// Mitsubishi GX Works2 project: exam_practice   PLC: Q02/Q02H

PROGRAM Q5-MC
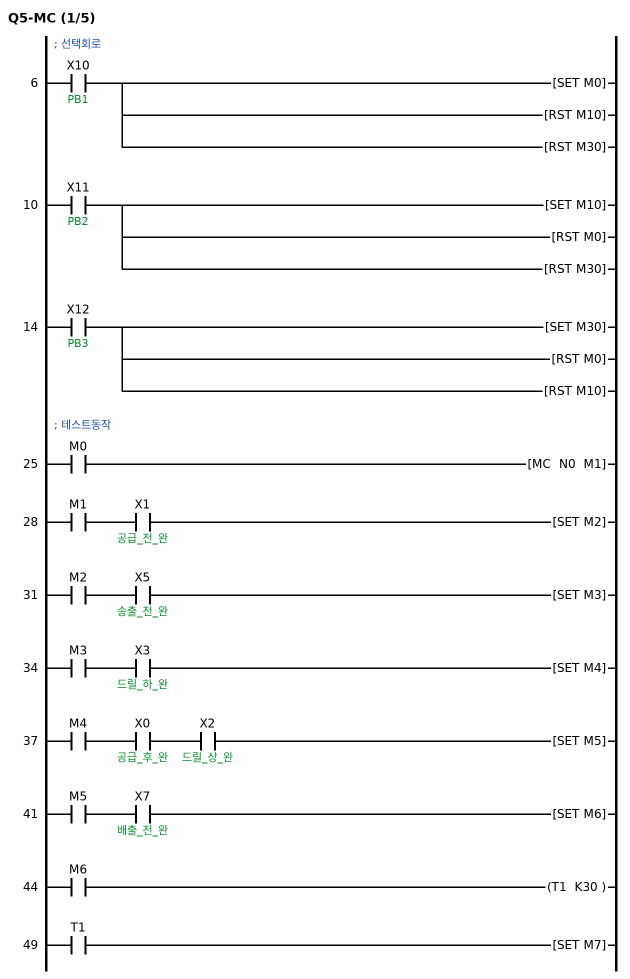
; 선택회로
6     LD      X10  ; PB1
      SET     M0
      RST     M10
      RST     M30
10    LD      X11  ; PB2
      SET     M10
      RST     M0
      RST     M30
14    LD      X12  ; PB3
      SET     M30
      RST     M0
      RST     M10
; 테스트동작
25    LD      M0
      MC      N0 M1
28    LD      M1
      AND     X1  ; 공급_전_완
      SET     M2
31    LD      M2
      AND     X5  ; 송출_전_완
      SET     M3
34    LD      M3
      AND     X3  ; 드릴_하_완
      SET     M4
37    LD      M4
      AND     X0  ; 공급_후_완
      AND     X2  ; 드릴_상_완
      SET     M5
41    LD      M5
      AND     X7  ; 배출_전_완
      SET     M6
44    LD      M6
      OUT     T1 K30
49    LD      T1
      SET     M7
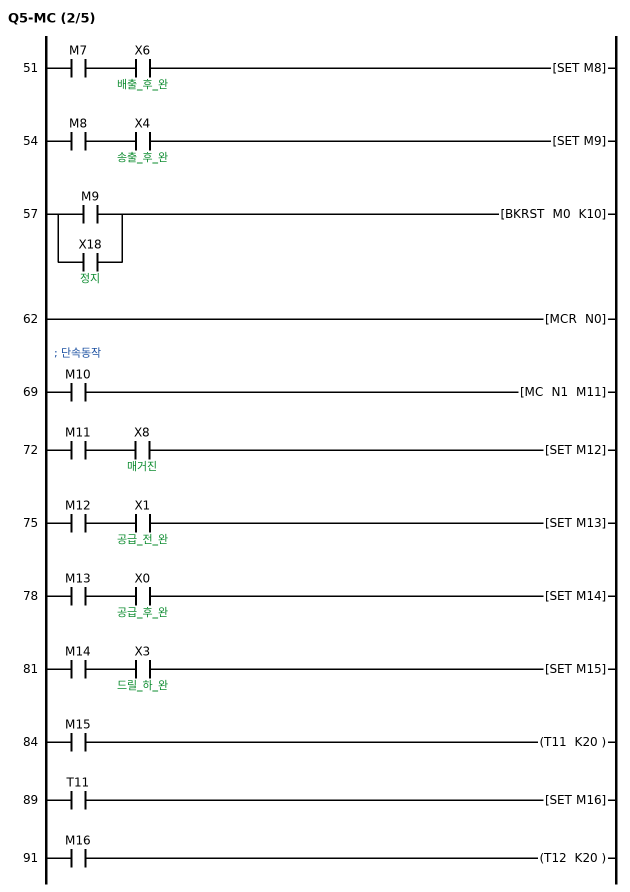
51    LD      M7
      AND     X6  ; 배출_후_완
      SET     M8
54    LD      M8
      AND     X4  ; 송출_후_완
      SET     M9
57    LD      M9
      OR      X18  ; 정지
      BKRST   M0 K10
62    MCR     N0
; 단속동작
69    LD      M10
      MC      N1 M11
72    LD      M11
      AND     X8  ; 매거진
      SET     M12
75    LD      M12
      AND     X1  ; 공급_전_완
      SET     M13
78    LD      M13
      AND     X0  ; 공급_후_완
      SET     M14
81    LD      M14
      AND     X3  ; 드릴_하_완
      SET     M15
84    LD      M15
      OUT     T11 K20
89    LD      T11
      SET     M16
91    LD      M16
      OUT     T12 K20
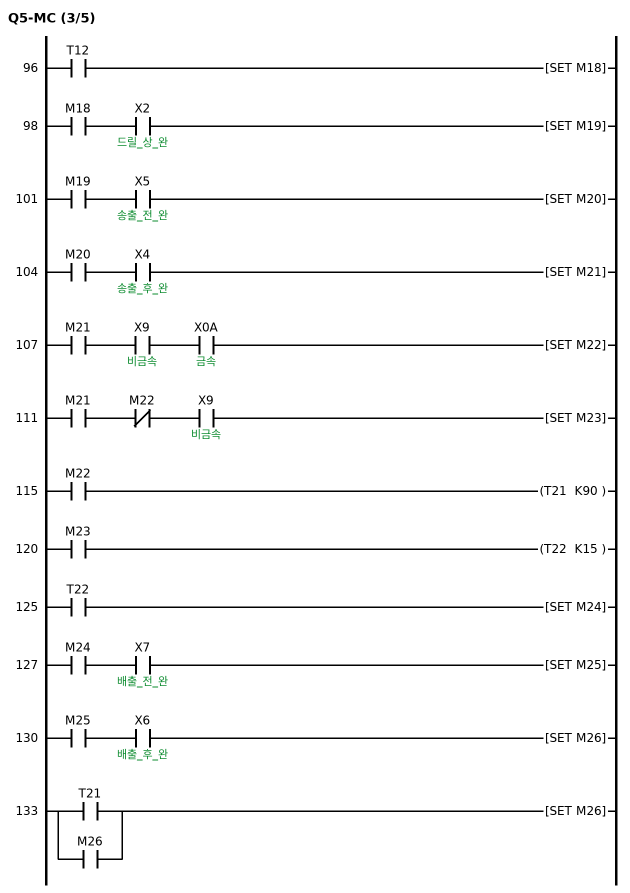
96    LD      T12
      SET     M18
98    LD      M18
      AND     X2  ; 드릴_상_완
      SET     M19
101   LD      M19
      AND     X5  ; 송출_전_완
      SET     M20
104   LD      M20
      AND     X4  ; 송출_후_완
      SET     M21
107   LD      M21
      AND     X9  ; 비금속
      AND     X0A  ; 금속
      SET     M22
111   LD      M21
      ANI     M22
      AND     X9  ; 비금속
      SET     M23
115   LD      M22
      OUT     T21 K90
120   LD      M23
      OUT     T22 K15
125   LD      T22
      SET     M24
127   LD      M24
      AND     X7  ; 배출_전_완
      SET     M25
130   LD      M25
      AND     X6  ; 배출_후_완
      SET     M26
133   LD      T21
      OR      M26
      SET     M26
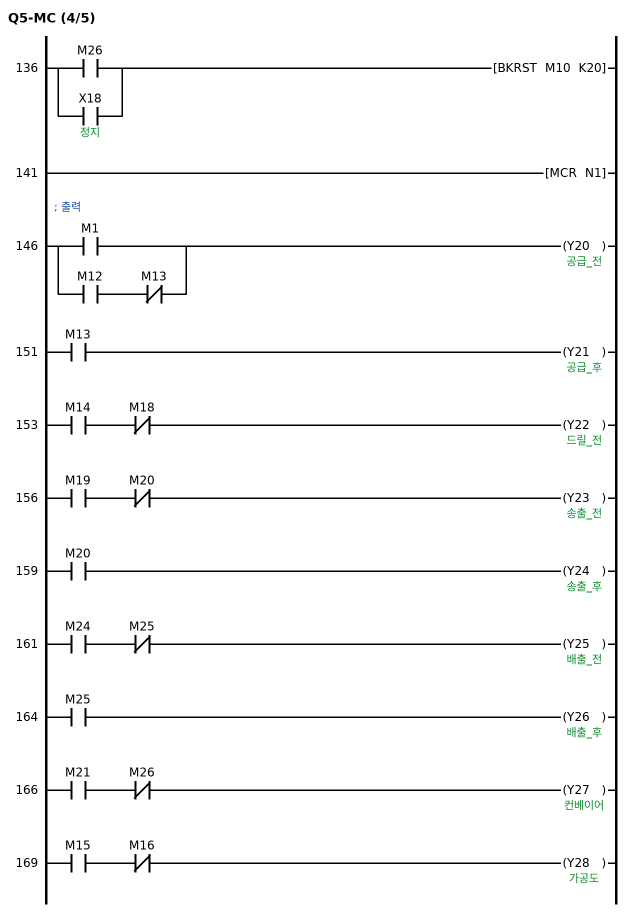
136   LD      M26
      OR      X18  ; 정지
      BKRST   M10 K20
141   MCR     N1
; 출력
146   LD      M1
      LD      M12
      ANI     M13
      ORB
      OUT     Y20  ; 공급_전
151   LD      M13
      OUT     Y21  ; 공급_후
153   LD      M14
      ANI     M18
      OUT     Y22  ; 드릴_전
156   LD      M19
      ANI     M20
      OUT     Y23  ; 송출_전
159   LD      M20
      OUT     Y24  ; 송출_후
161   LD      M24
      ANI     M25
      OUT     Y25  ; 배출_전
164   LD      M25
      OUT     Y26  ; 배출_후
166   LD      M21
      ANI     M26
      OUT     Y27  ; 컨베이어
169   LD      M15
      ANI     M16
      OUT     Y28  ; 가공도
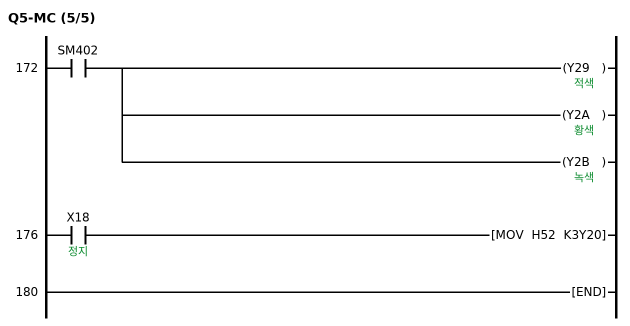
172   LD      SM402
      OUT     Y29  ; 적색
      OUT     Y2A  ; 황색
      OUT     Y2B  ; 녹색
176   LD      X18  ; 정지
      MOV     H52 K3Y20
180   END
END_PROGRAM
